{attribute 'qualified_only'}
// BOOL: True/False

VAR_GLOBAL
	
	// Control Enables
	bEnablePID 		: BOOL; // Enable PID Control
	bEnableFF 		: BOOL; // Enable FeedForward	
	bEnablePFB		: BOOL; // Enable Pressure Feedback
	bEnableU 		: BOOL; // Enable Signal to Valve

	bCharTesting	: BOOL; // Enable Characteristic testing
	bMove2Home		: BOOL; // Enable Home-function
	
	// No Function
	bEnableComp 	: BOOL; // Driving with Compensator
	
	// Enumerators
	nModeSelect		: E_Motion; // Motion Reference
	
END_VAR

(* stored: Version 1.1.0.1
   GVL G_Enables: Id {e1def63d-3986-47c4-8643-415c35f39ef1} *)
